SYSTEM test_CLIENT_SERVER2
  (* Version 1.0, 2023-10-23, Franz Höpfinger *)
  PACKAGE Training_CLIENT_SERVER;
  IMPORT VV::const::Computers::myComputers::C_PC_CLIENT;
  IMPORT VV::const::Computers::myComputers::C_PC_SERVER;
  IMPORT VV::const::ports::myPorts::PORT_A0;
  IMPORT VV::const::ports::myPorts::PORT_A1;
  IMPORT VV::const::ports::myPorts::PORT_A2;
  IMPORT VV::const::ports::myPorts::PORT_A3;
  IMPORT VV::const::ports::myPorts::PORT_B0;
  IMPORT VV::const::ports::myPorts::PORT_B1;
  IMPORT VV::const::ports::myPorts::PORT_B2;
  IMPORT VV::const::ports::myPorts::PORT_B3;
  IMPORT logiBUS::io::DI::logiBUS_DI::Input_I1;
  IMPORT logiBUS::io::DI::logiBUS_DI::Input_I2;
  IMPORT logiBUS::io::DI::logiBUS_DI::Input_I3;
  IMPORT logiBUS::io::DI::logiBUS_DI::Input_I4;
  IMPORT logiBUS::io::DQ::logiBUS_DO::Output_Q1;
  IMPORT logiBUS::io::DQ::logiBUS_DO::Output_Q2;
  IMPORT logiBUS::io::DQ::logiBUS_DO::Output_Q3;
  IMPORT logiBUS::io::DQ::logiBUS_DO::Output_Q4;
  APPLICATION App_CLIENT_SERVER
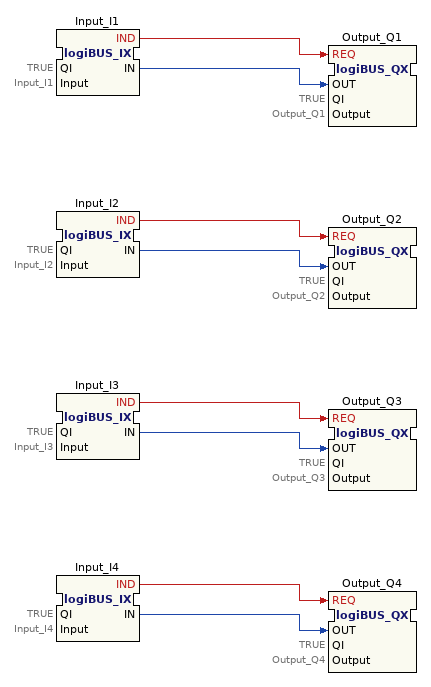
    FBS
      Input_I3 : logiBUS::io::DI::logiBUS_IX(QI := TRUE, Input := Input_I3);
      Input_I2 : logiBUS::io::DI::logiBUS_IX(QI := TRUE, Input := Input_I2);
      Input_I4 : logiBUS::io::DI::logiBUS_IX(QI := TRUE, Input := Input_I4);
      Output_Q2 : logiBUS::io::DQ::logiBUS_QX(QI := TRUE, Output := Output_Q2);
      Output_Q4 : logiBUS::io::DQ::logiBUS_QX(QI := TRUE, Output := Output_Q4);
      Output_Q3 : logiBUS::io::DQ::logiBUS_QX(QI := TRUE, Output := Output_Q3);
      Input_I1 : logiBUS::io::DI::logiBUS_IX(QI := TRUE, Input := Input_I1);
      Output_Q1 : logiBUS::io::DQ::logiBUS_QX(QI := TRUE, Output := Output_Q1);
    END_FBS
    EVENT_CONNECTIONS
      Input_I3.IND TO Output_Q3.REQ;
      Input_I2.IND TO Output_Q2.REQ;
      Input_I4.IND TO Output_Q4.REQ;
      Input_I1.IND TO Output_Q1.REQ;
    END_CONNECTIONS
    DATA_CONNECTIONS
      Input_I3.IN TO Output_Q3.OUT;
      Input_I2.IN TO Output_Q2.OUT;
      Input_I4.IN TO Output_Q4.OUT;
      Input_I1.IN TO Output_Q1.OUT;
    END_CONNECTIONS
  END_APPLICATION
  DEVICE FORTE_PC_CLIENT : iec61499::system::FORTE_PC(MGR_ID := C_PC_CLIENT (* Device manager socket ID *))
    {SET_ATTRIBUTE(Profile, HOLOBLOC)}
    RESOURCE EMB_RES_CLIENT : iec61499::system::EMB_RES
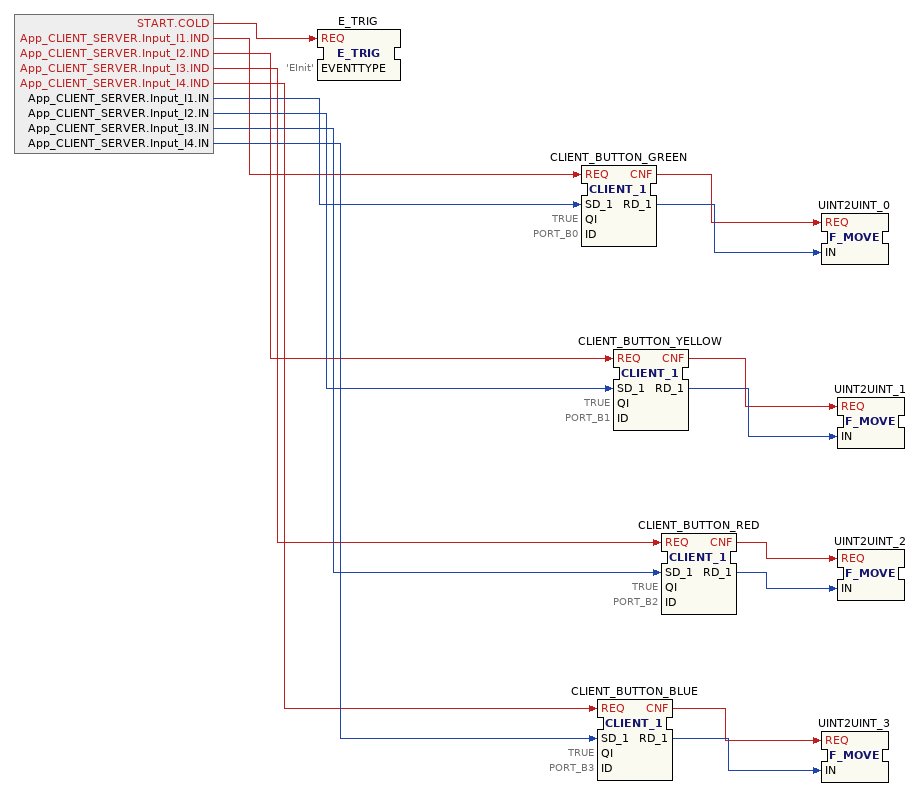
      FBS
        CLIENT_BUTTON_GREEN : iec61499::net::CLIENT_1(QI := TRUE, ID := PORT_B0);
        CLIENT_BUTTON_YELLOW : iec61499::net::CLIENT_1(QI := TRUE, ID := PORT_B1);
        CLIENT_BUTTON_RED : iec61499::net::CLIENT_1(QI := TRUE, ID := PORT_B2);
        CLIENT_BUTTON_BLUE : iec61499::net::CLIENT_1(QI := TRUE, ID := PORT_B3);
        UINT2UINT_0 : iec61131::selection::F_MOVE; {SET_ATTRIBUTE(DataType, UINT)}
        UINT2UINT_1 : iec61131::selection::F_MOVE; {SET_ATTRIBUTE(DataType, UINT)}
        UINT2UINT_2 : iec61131::selection::F_MOVE; {SET_ATTRIBUTE(DataType, UINT)}
        UINT2UINT_3 : iec61131::selection::F_MOVE; {SET_ATTRIBUTE(DataType, UINT)}
        E_TRIG : iec61499::events::E_TRIG(EVENTTYPE := 'EInit');
      END_FBS
      EVENT_CONNECTIONS
        CLIENT_BUTTON_GREEN.CNF TO UINT2UINT_0.REQ;
        CLIENT_BUTTON_RED.CNF TO UINT2UINT_2.REQ;
        CLIENT_BUTTON_YELLOW.CNF TO UINT2UINT_1.REQ;
        CLIENT_BUTTON_BLUE.CNF TO UINT2UINT_3.REQ;
        START.COLD TO E_TRIG.REQ;
        App_CLIENT_SERVER.Input_I1.IND TO CLIENT_BUTTON_GREEN.REQ;
        App_CLIENT_SERVER.Input_I2.IND TO CLIENT_BUTTON_YELLOW.REQ;
        App_CLIENT_SERVER.Input_I3.IND TO CLIENT_BUTTON_RED.REQ;
        App_CLIENT_SERVER.Input_I4.IND TO CLIENT_BUTTON_BLUE.REQ;
      END_CONNECTIONS
      DATA_CONNECTIONS
        CLIENT_BUTTON_GREEN.RD_1 TO UINT2UINT_0.IN;
        CLIENT_BUTTON_RED.RD_1 TO UINT2UINT_2.IN;
        CLIENT_BUTTON_YELLOW.RD_1 TO UINT2UINT_1.IN;
        CLIENT_BUTTON_BLUE.RD_1 TO UINT2UINT_3.IN;
        App_CLIENT_SERVER.Input_I1.IN TO CLIENT_BUTTON_GREEN.SD_1;
        App_CLIENT_SERVER.Input_I2.IN TO CLIENT_BUTTON_YELLOW.SD_1;
        App_CLIENT_SERVER.Input_I3.IN TO CLIENT_BUTTON_RED.SD_1;
        App_CLIENT_SERVER.Input_I4.IN TO CLIENT_BUTTON_BLUE.SD_1;
      END_CONNECTIONS
    END_RESOURCE
  END_DEVICE
  DEVICE FORTE_PC_SERVER : iec61499::system::FORTE_PC(MGR_ID := C_PC_SERVER (* Device manager socket ID *))
    {SET_ATTRIBUTE(Profile, HOLOBLOC)}
    RESOURCE EMB_RES_SERVER : iec61499::system::EMB_RES
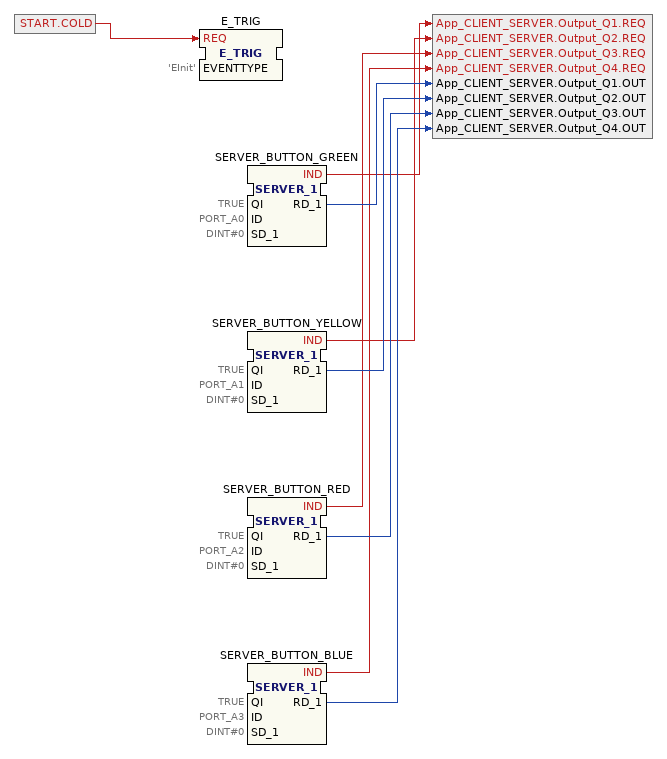
      FBS
        SERVER_BUTTON_GREEN : iec61499::net::SERVER_1(QI := TRUE, ID := PORT_A0, SD_1 := DINT#0);
        SERVER_BUTTON_RED : iec61499::net::SERVER_1(QI := TRUE, ID := PORT_A2, SD_1 := DINT#0);
        SERVER_BUTTON_YELLOW : iec61499::net::SERVER_1(QI := TRUE, ID := PORT_A1, SD_1 := DINT#0);
        SERVER_BUTTON_BLUE : iec61499::net::SERVER_1(QI := TRUE, ID := PORT_A3, SD_1 := DINT#0);
        E_TRIG : iec61499::events::E_TRIG(EVENTTYPE := 'EInit');
      END_FBS
      EVENT_CONNECTIONS
        START.COLD TO E_TRIG.REQ;
        SERVER_BUTTON_GREEN.IND TO App_CLIENT_SERVER.Output_Q1.REQ;
        SERVER_BUTTON_YELLOW.IND TO App_CLIENT_SERVER.Output_Q2.REQ;
        SERVER_BUTTON_RED.IND TO App_CLIENT_SERVER.Output_Q3.REQ;
        SERVER_BUTTON_BLUE.IND TO App_CLIENT_SERVER.Output_Q4.REQ;
      END_CONNECTIONS
      DATA_CONNECTIONS
        SERVER_BUTTON_GREEN.RD_1 TO App_CLIENT_SERVER.Output_Q1.OUT;
        SERVER_BUTTON_YELLOW.RD_1 TO App_CLIENT_SERVER.Output_Q2.OUT;
        SERVER_BUTTON_RED.RD_1 TO App_CLIENT_SERVER.Output_Q3.OUT;
        SERVER_BUTTON_BLUE.RD_1 TO App_CLIENT_SERVER.Output_Q4.OUT;
      END_CONNECTIONS
    END_RESOURCE
  END_DEVICE
  MAPPINGS
    App_CLIENT_SERVER.Input_I4 ON FORTE_PC_CLIENT.EMB_RES_CLIENT;
    App_CLIENT_SERVER.Input_I3 ON FORTE_PC_CLIENT.EMB_RES_CLIENT;
    App_CLIENT_SERVER.Input_I2 ON FORTE_PC_CLIENT.EMB_RES_CLIENT;
    App_CLIENT_SERVER.Output_Q3 ON FORTE_PC_SERVER.EMB_RES_SERVER;
    App_CLIENT_SERVER.Output_Q2 ON FORTE_PC_SERVER.EMB_RES_SERVER;
    App_CLIENT_SERVER.Output_Q4 ON FORTE_PC_SERVER.EMB_RES_SERVER;
    App_CLIENT_SERVER.Output_Q1 ON FORTE_PC_SERVER.EMB_RES_SERVER;
    App_CLIENT_SERVER.Input_I1 ON FORTE_PC_CLIENT.EMB_RES_CLIENT;
  END_MAPPINGS
END_SYSTEM
